TYPE Bits_VoltageRegulation_EAP :
STRUCT
	//Voltage Regulation
		Enable_VoltageRegulation : BIT;					//0
		Delta_Power_Limitation_VoltReg : BIT;			//1
		Enable_deadBandV : BIT;					//2
		Reset_To_Default_VoltReg : BIT;			//3
		Reserved1 : BIT;							//4
		Reserved2 : BIT;							//5
		Reserved3 : BIT;							//6
		Reserved4 : BIT;							//7
		Reserved5 : BIT;							//8
		Reserved6 : BIT;							//9
		Reserved7 : BIT;							//10
		Reserved8 : BIT;							//11
		Reserved9 : BIT;							//12
		Reserved10 : BIT;							//13
		Reserved11 : BIT;							//14
		Reserved12 : BIT;							//15
END_STRUCT
END_TYPE

(* stored: Version 1.1.0.1, ProductVersion 3.1.4022.18
   DUT Bits_VoltageRegulation_EAP: Id {68bef695-64cc-44bc-853b-d45d034508e1} *)
